TYPE ST_Selector :
STRUCT

	(* Meta info *)
	iId	: INT;	// Used to ID the selector attached to the system
	(* iId: Implemented to support switching selectors on the fly,
	the ID tells us which flow meter code to use, as the M2
	used several different flowmeters. *)

	(* Flowmeter *)
	(* Declare a structure for every possible FM *)
		
	
	//Common parameters

	(* Selector EPICS controls *)
    {attribute 'pytmc' := '
        pv: ValvesLockRequest
        io: io
     '}
	xResLock	:	BOOL; // request to lock the valves
    {attribute 'pytmc' := '
        pv: ValvesUnlockRequest
        io: io
     '}
	xResUnlock	:	BOOL; // request to unlock the valves
    {attribute 'pytmc' := '
        pv: ValvesLocked
        io: io
     '}
	xResLocked	:	BOOL; // valve movement is locked
    {attribute 'pytmc' := '
        pv: ValvesSynced
        io: io
     '}
	xResSyncd	:	BOOL; // valves are on the same position
    {attribute 'pytmc' := '
        pv: ValveSyncReqPos
        io: io
     '}
	iSyncReqPos	:	INT;  // requested position when synced
    {attribute 'pytmc' := '
        pv: Valve:01:ReqPos
        io: io
     '}
	iVici1ReqPos : INT;   // requested position for Vici 1
    {attribute 'pytmc' := '
        pv: Valve:02:ReqPos
        io: io
     '}
	iVici2ReqPos : INT;   // requested position for Vici 2
    
    //Hardware control
	stViciVlvCtrl	: ARRAY[1..2] OF	ST_ViciControl;
	
	(* Selector EPICS Readbacks *)
    {attribute 'pytmc' := '
        pv: ValvesPos
        io: i
     '}
	iSyncResPos : INT;
    
    //Hardware readbacks
    {attribute 'pytmc' := '
        pv: Valve
     '}
	stViciVlvStatus	: ARRAY[1..2] OF	ST_ViciStatus;

END_STRUCT
END_TYPE

(* stored: Version 1.1.0.1, ProductVersion 3.1.4024.2
   DUT ST_Selector: Id {edea215a-6843-498f-9e8b-ebe30f5a62c3} *)
